FUNCTION_BLOCK FB_ProbeRecipeCatalog EXTENDS FB_LocalRecipeProvider

;

METHOD M_ResetFixture
// This seam belongs only to the isolated TcUnit image, never production.
_catalog.SchemaVersion := 1;
_catalog.Count := 0;
_catalogInitialized := FALSE;
_catalogRestoreVersion := 0;
_n := 0;
END_METHOD

END_FUNCTION_BLOCK

(* stored: Version 1.1.0.1, ProductVersion 3.1.4024.12
   POU FB_ProbeRecipeCatalog: Id {0181356d-9ddb-467c-abe6-a4b8f92ad779}, SpecialFunc None
   Method M_ResetFixture: Id {49effafe-c58d-4797-b43e-b5429c654481} *)
